FUNCTION_BLOCK FB_LoadRecipe
VAR_INPUT
	sFileName : STRING(255); // Ex: 'C:\TwinCAT\Recipes\NomeDaReceita.json'
    bExecute  : BOOL;
END_VAR
VAR_OUTPUT
	bBusy   : BOOL;
    bDone   : BOOL;
    bError  : BOOL;
    nErrId  : UDINT;
END_VAR
VAR
	fbFileOpen  : FB_FileOpen;
    fbFileRead  : FB_FileRead;
    fbFileClose : FB_FileClose;
    fbJson      : FB_JsonDomParser;

    hFile    : UINT;
    sBuffer  : STRING(8192);
    jsonRoot : SJsonValue;
    jsonVal  : SJsonValue;
    idx      : INT;
    step     : INT;

    sPath    : STRING(255);
END_VAR

CASE step OF
0:
    IF bExecute THEN
        bBusy := TRUE;
        bDone := FALSE;
        bError := FALSE;
        nErrId := 0;

        fbFileOpen(
            sNetId := '',
            sPathName := sFileName,
            nMode := FOPEN_MODEREAD OR FOPEN_MODETEXT,
            bExecute := TRUE
        );

        step := 10;
    END_IF

10:
    fbFileOpen(bExecute := FALSE);
    IF NOT fbFileOpen.bBusy THEN
        IF fbFileOpen.bError THEN
            bError := TRUE;
            nErrId := fbFileOpen.nErrId;
            step := 100;
        ELSE
            hFile := fbFileOpen.hFile;
            fbFileRead(
                sNetId := '',
                hFile := hFile,
                pReadBuff := ADR(sBuffer),
                cbReadLen := SIZEOF(sBuffer),
                bExecute := TRUE
            );
            step := 20;
        END_IF
    END_IF

20:
    fbFileRead(bExecute := FALSE);
    IF NOT fbFileRead.bBusy THEN
        IF fbFileRead.bError THEN
            bError := TRUE;
            nErrId := fbFileRead.nErrId;
            step := 90;
        ELSE
            fbFileClose(sNetId := '', hFile := hFile, bExecute := TRUE);
            step := 30;
        END_IF
    END_IF

30:
    fbFileClose(bExecute := FALSE);
    IF NOT fbFileClose.bBusy THEN
        IF fbFileClose.bError THEN
            bError := TRUE;
            nErrId := fbFileClose.nErrId;
            step := 100;
        ELSE
            step := 40;
        END_IF
    END_IF

40:
    jsonRoot := fbJson.ParseDocument(sBuffer);
    IF jsonRoot = 0 THEN
        bError := TRUE;
        nErrId := 16#F1000001; // Código customizado para JSON inválido
        step := 100;
    ELSE
        step := 50;
    END_IF

50: //Fill the variables with Json buffer info [Parse Json file]
    sPath := 'stInfo/sMethodName';
    GVL_Recipe.stCurrentRecipe.stInfo.sMethodName := fbJson.GetString(fbJson.FindMemberPath(jsonRoot, sPath));

    sPath := 'stInfo/sCreatedBy';
    GVL_Recipe.stCurrentRecipe.stInfo.sCreatedBy := fbJson.GetString(fbJson.FindMemberPath(jsonRoot, sPath));

    sPath := 'stInfo/dCreationDate';
    GVL_Recipe.stCurrentRecipe.stInfo.dCreationDate := STRING_TO_DATE(fbJson.GetString(fbJson.FindMemberPath(jsonRoot, sPath)));

    sPath := 'stInfo/iRevision';
    GVL_Recipe.stCurrentRecipe.stInfo.iRevision := fbJson.GetInt(fbJson.FindMemberPath(jsonRoot, sPath));

    FOR idx := 1 TO 4 DO
        sPath := CONCAT('stSolventsTimes/aSolventN#', INT_TO_STRING(idx-1));
        GVL_Recipe.stCurrentRecipe.stSolventsTimes.aSolventN[idx] := TO_USINT(fbJson.GetInt(fbJson.FindMemberPath(jsonRoot, sPath)));

        sPath := CONCAT('stSolventsTimes/aTime#', INT_TO_STRING(idx-1));
        GVL_Recipe.stCurrentRecipe.stSolventsTimes.aTime[idx] := STRING_TO_TIME(fbJson.GetString(fbJson.FindMemberPath(jsonRoot, sPath)));

        sPath := CONCAT('stSolventsTimes/aVelocity#', INT_TO_STRING(idx-1));
        GVL_Recipe.stCurrentRecipe.stSolventsTimes.aVelocity[idx] := TO_INT(fbJson.GetInt(fbJson.FindMemberPath(jsonRoot, sPath)));
    END_FOR

    FOR idx := 1 TO 4 DO
        sPath := CONCAT('stVolumes/aT_IC_Volume#', INT_TO_STRING(idx-1));
        GVL_Recipe.stCurrentRecipe.stVolumes.aT_IC_Volume[idx] := LREAL_TO_REAL(fbJson.GetDouble(fbJson.FindMemberPath(jsonRoot, sPath)));
		
		sPath := CONCAT('stVolumes/aS0_Volume#', INT_TO_STRING(idx-1));
        GVL_Recipe.stCurrentRecipe.stVolumes.aS0_Volume[idx] := LREAL_TO_REAL(fbJson.GetDouble(fbJson.FindMemberPath(jsonRoot, sPath)));
		
		sPath := CONCAT('stVolumes/aS1_Volume#', INT_TO_STRING(idx-1));
        GVL_Recipe.stCurrentRecipe.stVolumes.aS1_Volume[idx] := LREAL_TO_REAL(fbJson.GetDouble(fbJson.FindMemberPath(jsonRoot, sPath)));
		
		sPath := CONCAT('stVolumes/aS2_Volume#', INT_TO_STRING(idx-1));
        GVL_Recipe.stCurrentRecipe.stVolumes.aS2_Volume[idx] := LREAL_TO_REAL(fbJson.GetDouble(fbJson.FindMemberPath(jsonRoot, sPath)));
		
		sPath := CONCAT('stVolumes/aS3_Volume#', INT_TO_STRING(idx-1));
        GVL_Recipe.stCurrentRecipe.stVolumes.aS3_Volume[idx] := LREAL_TO_REAL(fbJson.GetDouble(fbJson.FindMemberPath(jsonRoot, sPath)));
		
		sPath := CONCAT('stVolumes/aS4_Volume#', INT_TO_STRING(idx-1));
        GVL_Recipe.stCurrentRecipe.stVolumes.aS4_Volume[idx] := LREAL_TO_REAL(fbJson.GetDouble(fbJson.FindMemberPath(jsonRoot, sPath)));
		
		sPath := CONCAT('stVolumes/aS5_Volume#', INT_TO_STRING(idx-1));
        GVL_Recipe.stCurrentRecipe.stVolumes.aS5_Volume[idx] := LREAL_TO_REAL(fbJson.GetDouble(fbJson.FindMemberPath(jsonRoot, sPath)));
		
		sPath := CONCAT('stVolumes/aS6_Volume#', INT_TO_STRING(idx-1));
        GVL_Recipe.stCurrentRecipe.stVolumes.aS6_Volume[idx] := LREAL_TO_REAL(fbJson.GetDouble(fbJson.FindMemberPath(jsonRoot, sPath)));
		
		sPath := CONCAT('stVolumes/aS7_Volume#', INT_TO_STRING(idx-1));
        GVL_Recipe.stCurrentRecipe.stVolumes.aS7_Volume[idx] := LREAL_TO_REAL(fbJson.GetDouble(fbJson.FindMemberPath(jsonRoot, sPath)));
		
		sPath := CONCAT('stVolumes/aF_Volume#', INT_TO_STRING(idx-1));
        GVL_Recipe.stCurrentRecipe.stVolumes.aF_Volume[idx] := LREAL_TO_REAL(fbJson.GetDouble(fbJson.FindMemberPath(jsonRoot, sPath)));
		
    END_FOR

    sPath := 'stOtherParams/tSoakTime';
    GVL_Recipe.stCurrentRecipe.stOtherParams.tSoakTime := STRING_TO_TIME(fbJson.GetString(fbJson.FindMemberPath(jsonRoot, sPath)));
	
	sPath := 'stOtherParams/tAgitate1Time';
    GVL_Recipe.stCurrentRecipe.stOtherParams.tAgitate1Time := STRING_TO_TIME(fbJson.GetString(fbJson.FindMemberPath(jsonRoot, sPath)));
	
	sPath := 'stOtherParams/tAgitade2Time';
    GVL_Recipe.stCurrentRecipe.stOtherParams.tAgitade2Time := STRING_TO_TIME(fbJson.GetString(fbJson.FindMemberPath(jsonRoot, sPath)));
	
	sPath := 'stOtherParams/iVialsToFill';
    GVL_Recipe.stCurrentRecipe.stOtherParams.iVialsToFill := TO_USINT(fbJson.GetInt(fbJson.FindMemberPath(jsonRoot, sPath)));
	
	sPath := 'stOtherParams/rVialPrimeVol';
    GVL_Recipe.stCurrentRecipe.stOtherParams.rVialPrimeVol := LREAL_TO_REAL(fbJson.GetDouble(fbJson.FindMemberPath(jsonRoot, sPath)));
	
	sPath := 'stOtherParams/rVial1FillVol';
    GVL_Recipe.stCurrentRecipe.stOtherParams.rVial1FillVol := LREAL_TO_REAL(fbJson.GetDouble(fbJson.FindMemberPath(jsonRoot, sPath)));
	
	sPath := 'stOtherParams/rVials2_4FillVol';
    GVL_Recipe.stCurrentRecipe.stOtherParams.rVials2_4FillVol := LREAL_TO_REAL(fbJson.GetDouble(fbJson.FindMemberPath(jsonRoot, sPath)));
	
	sPath := 'stOtherParams/tAirDryTime';
    GVL_Recipe.stCurrentRecipe.stOtherParams.tAirDryTime := STRING_TO_TIME(fbJson.GetString(fbJson.FindMemberPath(jsonRoot, sPath)));

    step := 100;

90:
    fbFileClose(sNetId := '', hFile := hFile, bExecute := TRUE);
    step := 100;

100:
    bBusy := FALSE;
    bDone := NOT bError;
    IF NOT bExecute THEN
        step := 0;
    END_IF
END_CASE

END_FUNCTION_BLOCK

(* stored: Version 1.1.0.1, ProductVersion 3.1.4024.12
   POU FB_LoadRecipe: Id {fdbedb76-49e0-47f1-8b40-c95081ed8fdc}, SpecialFunc None *)
